// Axis Errors -----------------------------------------------------------------------------------------------------


17152   : sNcError := '17152 Parameter: Axis ID not allowed. The axis ID value is not allowed, e.g. because it has already been assigned, is out of the valid range [1 ... 255], or does not exist in the current configuration.';
17153   : sNcError := '17153 Parameter: Axis type not allowed. The axis type value is not allowed as it is not defined. Valid types: 1 (servo), 2 (fast/creep), 3 (stepper motor).';
17158   : sNcError := '17158 Parameter: Slow manual velocity not allowed. The slow manual velocity value is not allowed. Valid range: [0.0, 10000.0] e.g., m/min.';
17159   : sNcError := '17159 Parameter: Fast manual velocity not allowed. The fast manual velocity value is not allowed. Valid range: [0.0, 10000.0] e.g., m/min.';
17160   : sNcError := '17160 Parameter: Rapid traverse velocity not allowed. The rapid traverse velocity value is not allowed. Valid range: [0.0, 10000.0] e.g., m/min.';
17161   : sNcError := '17161 Parameter: Axis acceleration not allowed. The axis acceleration value is not allowed. Valid range: [0.0, 1000000.0] e.g., m/s².';
17162   : sNcError := '17162 Parameter: Axis deceleration not allowed. The axis deceleration value is not allowed. Valid range: [0.0, 1000000.0] e.g., m/s².';
17163   : sNcError := '17163 Parameter: Axis jerk not allowed. The axis jerk value is not allowed. Valid range: [0.0, 1000000.0] e.g., m/s³.';
17164   : sNcError := '17164 Parameter: Delay time between position and velocity not allowed. The delay time for dead time compensation is not allowed. Valid range: [0, 0.1] s.';
17165   : sNcError := '17165 Parameter: Override type not allowed. The velocity override type value is not allowed as it is not defined. Valid types: 1 (internal), 2 (external).';
17166   : sNcError := '17166 Parameter: NCI: Velo-Jump-Factor not allowed. The velo-jump-factor value is not allowed for TwinCAT NCI. Valid range: [0, 1000000].';
17167   : sNcError := '17167 Parameter: NCI: Tolerance sphere radius invalid. The tolerance sphere size value for auxiliary axes is invalid. Valid range: [0, 1000] e.g., mm.';
17168   : sNcError := '17168 Parameter: NCI: Max deviation for auxiliary axis invalid. The max allowed deviation value for auxiliary axes is invalid. Valid range: [0, 10000] e.g., mm.';
17170   : sNcError := '17170 Parameter: Referencing velocity in direction of cam not allowed. The referencing velocity towards the cam is not allowed. Valid range: [0.0, 10000.0] e.g., m/min.';
17171   : sNcError := '17171 Parameter: Referencing velocity in sync direction not allowed. The referencing velocity towards the sync pulse is not allowed. Valid range: [0.0, 10000.0] e.g., m/min.';
17172   : sNcError := '17172 Parameter: Pulse width in positive direction not allowed. The pulse width in the positive direction is not allowed for pulsed operation. Valid range: [0.0, 1000000.0] e.g., mm.';
17173   : sNcError := '17173 Parameter: Pulse width in negative direction not allowed. The pulse width in the negative direction is not allowed for pulsed operation. Valid range: [0.0, 1000000.0] e.g., mm.';
17174   : sNcError := '17174 Parameter: Pulse time in positive direction not allowed. The pulse time in the positive direction is not allowed. Valid range: [0.0, 600.0] s.';
17175   : sNcError := '17175 Parameter: Pulse time in negative direction not allowed. The pulse time in the negative direction is not allowed. Valid range: [0.0, 600.0] s.';
17176   : sNcError := '17176 Parameter: Creep distance in positive direction not allowed. The creep distance in the positive direction is not allowed. Valid range: [0.0, 100000.0] e.g., mm.';
17177   : sNcError := '17177 Parameter: Creep distance in negative direction not allowed. The creep distance in the negative direction is not allowed. Valid range: [0.0, 100000.0] e.g., mm.';
17178   : sNcError := '17178 Parameter: Braking distance in positive direction not allowed. The braking distance in the positive direction is not allowed. Valid range: [0.0, 100000.0] e.g., mm.';
17179   : sNcError := '17179 Parameter: Braking distance in negative direction not allowed. The braking distance in the negative direction is not allowed. Valid range: [0.0, 100000.0] e.g., mm.';
17180   : sNcError := '17180 Parameter: Deceleration time in positive direction not allowed. The deceleration time in the positive direction is not allowed. Valid range: [0.0, 60.0] s.';
17181   : sNcError := '17181 Parameter: Deceleration time in negative direction not allowed. The deceleration time in the negative direction is not allowed. Valid range: [0.0, 60.0] s.';
17182   : sNcError := '17182 Parameter: Switching time from rapid to slow traverse not allowed. The switching time from rapid to slow traverse is not allowed. Valid range: [0.0, 60.0] s.';
17183   : sNcError := '17183 Parameter: Creep distance for stop not allowed. The creep distance for an explicit stop is not allowed. Valid range: [0.0, 100000.0] e.g., mm.';
17184   : sNcError := '17184 Parameter: Motion monitoring not allowed. The motion monitoring activation value is not allowed. Valid range: [0, 1].';
17185   : sNcError := '17185 Parameter: Position window monitoring not allowed. The position window monitoring activation value is not allowed. Valid range: [0, 1].';
17186   : sNcError := '17186 Parameter: Target window monitoring not allowed. The target window monitoring activation value is not allowed. Valid range: [0, 1].';
17187   : sNcError := '17187 Parameter: Loop not allowed. The loop movement activation value is not allowed. Valid range: [0, 1].';
17188   : sNcError := '17188 Parameter: Motion monitoring time not allowed. The motion monitoring time value is not allowed. Valid range: [0.0, 600.0] s.';
17189   : sNcError := '17189 Parameter: Target window range not allowed. The target window value is not allowed. Valid range: [0.0, 10000.0] e.g., mm.';
17190   : sNcError := '17190 Parameter: Position window range not allowed. The position window value is not allowed. Valid range: [0.0, 10000.0] e.g., mm.';
17191   : sNcError := '17191 Parameter: Position window monitoring time not allowed. The position window monitoring time value is not allowed. Valid range: [0.0, 600.0] s.';
17192   : sNcError := '17192 Parameter: Looping distance not allowed. The looping distance value is not allowed. Valid range: [0.0, 10000.0] e.g., mm.';
17193   : sNcError := '17193 Parameter: Axis cycle time not allowed. The axis cycle time value is not allowed. Valid range: [0.001, 0.1] s.';
17194   : sNcError := '17194 Parameter: Operation mode stepper motor not allowed. The stepper motor operating mode value is not allowed. Valid range: [1, 2].';
17195   : sNcError := '17195 Parameter: Displacement per stepper motor step not allowed. The displacement per step value for the stepper motor is not allowed. Valid range: [0.000001, 1000.0] e.g., mm/STEP.';
17196   : sNcError := '17196 Parameter: Minimum velocity for stepper motor set value profile not allowed. The minimum velocity for the stepper motor velocity profile is not allowed. Valid range: [0.0, 1000.0] e.g., m/min.';
17197   : sNcError := '17197 Parameter: Stepper motor stages for one velocity level not allowed. The number of steps for each velocity level in the setpoint generation is not allowed. Valid range: [0, 100].';
17198   : sNcError := '17198 Parameter: DWORD for the interpretation of the axis units not allowed. The flags value for interpreting position and velocity units is not allowed. Valid range: [0, 0xFFFFFFFF].';
17199   : sNcError := '17199 Parameter: Maximum velocity not allowed. The maximum permitted velocity value is not allowed. Valid range: [0.0, 10000.0] e.g., m/min.';
17200   : sNcError := '17200 Parameter: Motion monitoring window not allowed. The motion monitoring window value is not allowed. Valid range: [0.0, 10000.0] e.g., mm.';
17201   : sNcError := '17201 Parameter: PEH time monitoring not allowed. The PEH time monitoring activation value is not allowed (PEH: positioning end and halt). Valid range: [0, 1].';
17202   : sNcError := '17202 Parameter: PEH monitoring time not allowed. The PEH monitoring time (timeout) value is not allowed (PEH: positioning end and halt). Valid range: [0.0, 600.0] s.';
17203   : sNcError := '17203 Parameter: Brake Release Delay is invalid. The brake release delay parameter for a rapid/slow traverse axis is invalid. Valid range: [0.0, 60.0] s.';
17204   : sNcError := '17204 Parameter: NC Data Persistence is invalid. The boolean parameter NC Data Persistence of an axis is invalid. Valid range: [0, 1].';
17205   : sNcError := '17205 Parameter: Error reaction mode is invalid. The error reaction mode parameter of the axis is invalid (instantaneous, delayed). Valid range: [0, 1].';
17206   : sNcError := '17206 Parameter: Error reaction delay is invalid. The error reaction delay parameter of the axis is invalid. Valid range: [0.0, 1000.0] s.';
17207   : sNcError := '17207 Parameter: Use actual values in deactivated state is invalid. The parameter "Use actual values in deactivated state" is invalid. Valid range: [0, 1].';
17208   : sNcError := '17208 Parameter: Allow motion commands for slave axes is invalid. The boolean parameter "Allow motion commands for slave axes" is invalid. Valid range: [0, 1].';
17209   : sNcError := '17209 Parameter: Allow motion commands for axis in external setpoint generation is invalid. The boolean parameter "Allow motion commands for axis in external setpoint generation" is invalid. Valid range: [0, 1].';
17210   : sNcError := '17210 Parameter: Fading Acceleration is invalid. The "Fading Acceleration" parameter for the fading profile from SET to ACTUAL values is invalid. Valid range: [0; 0.01 .. 1.0e+20] e.g., mm/s².';
17211   : sNcError := '17211 Parameter: Fast Axis Stop signal type not allowed. The Signal Type value of the "Fast Axis Stop" is not allowed. Valid range: [0...5].';
17212   : sNcError := '17212 Parameter: ADS index offset not allowed. The "ADS offset (axis state)" value for user-defined parameter named "UserData" in AxisRef is invalid.';
17216   : sNcError := '17216 Initialization: Axis initialization. The axis has not been fully initialized (I/O, axis, reset).';
17217   : sNcError := '17217 Address: Group address. The axis does not have a group or the group address has not been initialized.';
17218   : sNcError := '17218 Address: Encoder address. The axis does not have an encoder or the encoder address has not been initialized.';
17219   : sNcError := '17219 Address: Controller address. The axis does not have a controller or the controller address has not been initialized.';
17220   : sNcError := '17220 Address: Drive address. The axis does not have a drive or the drive address has not been initialized.';
17221   : sNcError := '17221 Address: Axis interface PLC to NC address. The axis has no axis interface from the PLC to the NC (PlcToNc) or the axis interface address has not been initialized.';


// Drive Errors -----------------------------------------------------------------------------------------------------


17920   : sNcError := '17920 Parameter: Drive ID not allowed. The drive ID value is invalid because it is either already assigned, less than or equal to zero, or exceeds 255. Valid range: [1 ... 255].';
17921   : sNcError := '17921 Parameter: Drive type not allowed. The drive type value is invalid as it is not defined. Valid range: [1, 20].';
17922   : sNcError := '17922 Parameter: Drive operation mode not allowed. The drive operation mode value is invalid. Valid range: [1].';
17923   : sNcError := '17923 Parameter: Motor polarity not allowed. The motor polarity flag is invalid. Valid values: 0 (Positive), 1 (Negative).';
17924   : sNcError := '17924 Parameter: Drift compensation/velocity offset (DAC offset) invalid. Valid range: [-100.0, 100.0] e.g., m/min.';
17925   : sNcError := '17925 Parameter: Reference velocity (velocity pre-control) invalid. Valid range: [0.0, 10000.0] e.g., m/min.';
17926   : sNcError := '17926 Parameter: Reference output in percent invalid. The value usually corresponds to a voltage of 10.0 V. Valid range: [0.0, 5.0] %.';
17927   : sNcError := '17927 Parameter: Quadrant compensation factor not allowed. The value is invalid. Valid range: [0.0, 100.0].';
17928   : sNcError := '17928 Parameter: Velocity reference point in percent invalid. The value 1.0 corresponds to 100 percent. Valid range: [0.01, 1.0] %.';
17929   : sNcError := '17929 Parameter: Output reference point invalid. The value 1.0 corresponds to 100 percent. Valid range: [0.01, 1.0] %.';
17930   : sNcError := '17930 Parameter: Min or max output limits (output limitation) invalid. The min limit is initially set to –1.0 (-100%) and the max limit to 1.0 (100%). Valid range: [-1.0, 1.0] %.';
17931   : sNcError := '17931 Parameter: Maximum value for output not allowed. The value for the max output digits of the drive is not allowed. Valid range: [0x000000FF .. 0xFFFFFFFF] INC or Digits.';
17932   : sNcError := '17932 Parameter: Internal Drive Control Word not allowed. The internal Drive Control Word value for the NC is invalid. Valid range: [>0].';
17933   : sNcError := '17933 Parameter: Internal timer for RESET behavior Drive not allowed. The timer influencing NC Drive and IO Drive behavior is invalid. Valid range: [>5] NC SEC cycles.';
17934   : sNcError := '17934 Parameter: Master Motion Controller ID not allowed. This parameter is invalid for a slave NC Motion Controller. Valid range: [0 .. 255].';
17935   : sNcError := '17935 Parameter: Drive torque output scaling not allowed. The value for Drive torque output scaling (rotary motor) or force output scaling (linear motor) is invalid. Valid range: [0, 1000000].';
17936   : sNcError := '17936 Parameter: Drive velocity output scaling not allowed. The value is invalid. Valid range: [0, 1000000].';
17937   : sNcError := '17937 Parameter: Profi Drive DSC proportional gain Kpc (controller) not allowed. The Profi Drive DSC position control gain (Kpc factor) value is invalid. Valid range: [0, 0xFFFFFF] 0.001 * 1/s.';
17938   : sNcError := '17938 Parameter: Table ID not allowed. The table ID value is invalid. Valid range: [0, 255].';
17939   : sNcError := '17939 Parameter: Table interpolation type not allowed. The table interpolation type value is invalid. Valid values: 0 (LINEAR), 2 (SPLINE).';
17940   : sNcError := '17940 Parameter: Output offset in percent not allowed. The output offset in percent value is invalid. Valid range: [-1.0, 1.0] %.';
17941   : sNcError := '17941 Parameter: Profi Drive DSC scaling for "Xerr" (controller) not allowed. The value is invalid. Valid range: [0, 1000000].';
17942   : sNcError := '17942 Parameter: Drive acceleration output scaling not allowed. The value is invalid. Valid range: [0, 1000000].';
17943   : sNcError := '17943 Parameter: Drive position output scaling not allowed. The value is invalid. Valid range: [0, 1000000].';
17944   : sNcError := '17944 Parameter: Dead time compensation mode (Motion Controller) invalid. The dead time compensation mode is invalid (OFF, ON with velocity, ON with velocity and acceleration). Valid values: [0, 1, 2].';
17945   : sNcError := '17945 Parameter: Control bits of dead time compensation (motion controller) invalid. The parameter is invalid. Valid range: [>0].';
17946   : sNcError := '17946 Parameter: Time shift of dead time compensation mode (motion controller) invalid. The time shift parameter in nanoseconds is invalid. Valid range: [-1.0E9 .. 1.0E9] ns.';
17947   : sNcError := '17947 Parameter: Output delay velocity interface Motion Controller invalid. The optional output delay in the velocity interface is invalid. Valid range: [0.0 .. 0.1] s.';
17948   : sNcError := '17948 Parameter: Drive filter type not allowed for command variable filter for the output position. The drive filter type value is invalid. Valid range: [0, 2].';
17949   : sNcError := '17949 Parameter: Drive filter time not allowed for command variable filter for the output position. The drive filter time value is invalid. Valid range: [0.0, 1.0] s.';
17950   : sNcError := '17950 Parameter: Drive filter order not allowed for command variable filter for the output position. The drive filter order value is invalid. Valid range: [0, 10].';
17952   : sNcError := '17952 Parameter: Bit mask for stepper motor cycle not allowed. The bit mask value is invalid. Valid range: [0, 255].';
17953   : sNcError := '17953 Parameter: Bit mask for stepper motor holding current not allowed. The holding current mask value is invalid. Valid range: [0, 255].';
17954   : sNcError := '17954 Parameter: Scaling factor for actual torque (actual current) not allowed. The scaling factor value is invalid. Valid range: [0, 1E+30].';
17955   : sNcError := '17955 Parameter: Filter time for actual torque not allowed. The filter time value for the actual torque (or current) is invalid. Valid range: [0.0, 60.0] s.';
17956   : sNcError := '17956 Parameter: Filter time for the time derivative of the actual torque not allowed. The filter time value for the time derivative of the actual torque (or current) is invalid. Valid range: [0.0, 60.0] s.';
17957   : sNcError := '17957 Parameter: Drive operation mode invalid. The drive operation mode parameter is invalid. Valid range: [0, >=1].';
17958   : sNcError := '17958 Monitoring: Motion Controller function not supported. The triggered Motion Controller functionality is not enabled or implemented.';
17959   : sNcError := '17959 Function: DRIVEOPERATIONMODEBUSY. The drive operation mode activation failed because another object is using this interface.';
17960   : sNcError := '17960 Monitoring: Drive operation mode changeover not configured. No drive operation mode changeover is configured or the desired mode is not found.';
17961   : sNcError := '17961 Monitoring: Feedback drive operation mode changeover. The requested drive operation mode was not consistently reported back within the monitoring time.';
17968   : sNcError := '17968 Monitoring: Overtemperature detected or reported in the drive or terminal.';
17969   : sNcError := '17969 Monitoring: Undervoltage detected or reported in the drive or terminal.';
17970   : sNcError := '17970 Monitoring: Wire break in phase A detected or reported in the drive or terminal.';
17971   : sNcError := '17971 Monitoring: Wire break in phase B detected or reported in the drive or terminal.';
17972   : sNcError := '17972 Monitoring: Overcurrent detected or reported in phase A in the drive or terminal.';
17973   : sNcError := '17973 Monitoring: Overcurrent detected or reported in phase B in the drive or terminal.';
17974   : sNcError := '17974 Monitoring: Torque overload (stall) detected or reported in the drive or terminal.';
17984   : sNcError := '17984 Initialization: Drive initialization. Drive not initialized properly. Steps: 1. Initialization drive I/O, 2. Initialization drive, 3. Reset drive.';
17985   : sNcError := '17985 Address: Axis address not initialized. The drive does not know its axis or the axis address is not initialized.';
17986   : sNcError := '17986 Address: Address I/O input structure. The drive has no valid I/O input address in the process image.';
17987   : sNcError := '17987 Address: Address I/O output structure. The drive has no valid I/O output address in the process image.';
18000   : sNcError := '18000 Monitoring: Drive hardware not ready. The drive hardware is not ready for operation, possibly due to hardware error, start-up phase, or missing controller enable.';
18001   : sNcError := '18001 Monitoring: Error in cyclic communication of the drive (Life Counter). Possible causes: interrupted fieldbus or drive in error state.';
18002   : sNcError := '18002 Monitoring: Changing table ID with active controller enable not allowed. Changing the characteristic curve table ID is not allowed when controller enable is active.';
18005   : sNcError := '18005 Monitoring: I/O data for more than "n" continuous NC cycles invalid. The axis detected invalid I/O data for more than "n" continuous NC cycles.';


// Controller Errors -----------------------------------------------------------------------------------------------------


17664   : sNcError := '17664 Parameter: Controller ID not allowed. The controller ID value is invalid, e.g., already assigned, less than or equal to zero, or exceeds 255. Valid range: [1 ... 255].';
17665   : sNcError := '17665 Parameter: Controller type not allowed. The controller type value is invalid as it is not defined. Valid types: 1 (P-controller), 7 (Fast/creep), 8 (Stepper motor), 9 (Sercos).';
17666   : sNcError := '17666 Parameter: Operation mode controller not allowed. The controller operating mode value is invalid. Valid range: [1].';
17667   : sNcError := '17667 Parameter: Weighting of the velocity pre-control not allowed. The velocity pre-control weighting value is invalid. Valid range: [0.0 ... 1.0] %.';
17668   : sNcError := '17668 Parameter: Lag error monitor (position) not allowed. The activation value for the lag error monitor is invalid. Valid range: [0, 1].';
17669   : sNcError := '17669 Parameter: Lag monitoring (velocity) not allowed. The activation value for the lag error monitoring is invalid. Valid range: [0, 1].';
17670   : sNcError := '17670 Parameter: Lag error window (position) not allowed. The maximum allowable lag error value is invalid. Valid range: [0.0, 10000.0] e.g., mm.';
17671   : sNcError := '17671 Parameter: Lag error filter time (position) not allowed. The lag error filter time value is invalid. Valid range: [0.0, 600.0] s.';
17672   : sNcError := '17672 Parameter: Lag error window (velocity) not allowed. The lag error window (velocity) value is invalid. Valid range: [0.0, 10000.0] e.g., m/min.';
17673   : sNcError := '17673 Parameter: Lag error filter time (velocity) not allowed. The lag error filter time value is invalid. Valid range: [0.0, 600.0] s.';
17674   : sNcError := '17674 Parameter: Controller output limitation not allowed. The output limitation value of the controller is invalid. Valid range: [0.0, 1.0] %.';
17680   : sNcError := '17680 Parameter: Proportional gain Kv or Kp (controller) not allowed. The proportional gain (Kv or Kp factor) value is invalid. Valid range: [0.0, 10000.0] e.g., mm/s/mm.';
17681   : sNcError := '17681 Parameter: Integral action time Tn (controller) not allowed. The integral action time value is invalid (I part of the PID T1 controller). Valid range: [0.0, 60.0] s.';
17682   : sNcError := '17682 Parameter: Rate time Tv (controller) not allowed. The derivative action time value is invalid (D part of the PID T1 controller). Valid range: [0.0, 60.0] s.';
17683   : sNcError := '17683 Parameter: Damping time Td (controller) not allowed. The damping time value is invalid (D part of the PID T1 controller). Valid range: [0.0, 60.0] s.';
17684   : sNcError := '17684 Function: Activation of the automatic offset calibration not allowed. Activation of automatic offset calibration is only possible for certain controllers (without I component).';
17685   : sNcError := '17685 Parameter: Additional proportional gain Kv or Kp (controller) not allowed. The second term of the proportional gain value is invalid. Valid range: [0.0, 10000.0] e.g., mm/s/mm.';
17686   : sNcError := '17686 Parameter: Reference velocity for additional proportional gain Kv or Kp (controller) not allowed. The reference velocity percentage value is invalid. Standard: 0.5 (50%). Valid range: [0.0 ... 1.0] %.';
17687   : sNcError := '17687 Parameter: Proportional gain Pa (proportion) not allowed. The proportional gain (Pa factor) value is invalid. Valid range: [0.0, 1000000.0] s.';
17688   : sNcError := '17688 Parameter: Proportional gain Kv (controller) not allowed. The proportional gain (Kv factor) value is invalid. Valid range: [0.0, 10000.0].';
17689   : sNcError := '17689 Parameter: Integral action time Tn (controller) not allowed. The integral action time value is invalid (I part of the PID T1 controller). Valid range: [0.0, 60.0] s.';
17690   : sNcError := '17690 Parameter: Reserved. Reserved, currently not used.';
17691   : sNcError := '17691 Parameter: Reserved. Reserved, currently not used.';
17692   : sNcError := '17692 Parameter: Velocity filter time not allowed. The velocity filter time in seconds (P-T1 filter) is invalid. Valid range: [0.0, 60.0] s.';
17693   : sNcError := '17693 Parameter: Dead range not allowed. The dead range (neutral zone) value of the position or velocity error is invalid. Valid range: [0.0, 10000.0] mm or mm/s.';
17695   : sNcError := '17695 Parameter: Proportional gain Kcp not allowed. The proportional gain Kcp parameter for slave coupling difference control is invalid. Valid range: [0.0, 10000.0] e.g., mm²/mm.';
17696   : sNcError := '17696 Parameter: Rate time Tv (controller) not allowed. The derivative action time value is invalid (D part of the PID T1 controller). Valid range: [0.0, 60.0] s.';
17697   : sNcError := '17697 Parameter: Damping time Td (controller) not allowed. The damping time value is invalid (D part of the PID T1 controller). Valid range: [0.0, 60.0] s.';
17698   : sNcError := '17698 Parameter: Limitation of the I part not allowed. The limitation parameter for the I-part of a PI- or PID-controller is invalid. Valid range: [0.0 .. 1.0] %.';
17699   : sNcError := '17699 Parameter: Limitation of the D part not allowed. The limitation parameter for the D-part of a PI- or PID-controller is invalid. Valid range: [0.0 .. 1.0] %.';
17700   : sNcError := '17700 Parameter: Deactivation of the I part during travel not allowed. The boolean parameter for switching off the I-part during active positioning is invalid. Valid range: [0, 1].';
17701   : sNcError := '17701 Parameter: Filter time for P-T2 filter not allowed. The filter time T0 for the P-T2 element is invalid. Valid range: [0.0, 60.0] s.';
17702   : sNcError := '17702 Parameter: Velocity observer mode not allowed. The parameterized mode (0=OFF, 1=LUENBERGER) for the velocity observer is invalid. Valid range: [0, 1].';
17703   : sNcError := '17703 Parameter: Motor torque constant Kt or Kf not allowed. The motor torque constant Kt (rotary) or Kf (linear) parameter for the velocity observer is invalid. Valid range: [0.0 .. 100000.0] Nm/A or N/A.';
17704   : sNcError := '17704 Parameter: Motor moment of inertia JM not allowed. The motor moment of inertia JM parameter for the velocity observer is invalid. Valid range: [0.0001 .. 100000.0] kg cm².';
17705   : sNcError := '17705 Parameter: Bandwidth f0 not allowed. The bandwidth f0 parameter for the velocity observer is invalid. Valid range: [0.0 .. 10000.0] Hz.';
17706   : sNcError := '17706 Parameter: Correction factor kc not allowed. The correction factor kc for the velocity observer is invalid. Valid range: [0.0 .. 100.0] s.';
17707   : sNcError := '17707 Parameter: Time constant T for 1st order filter not allowed. The time constant T for the 1st order velocity filter is invalid. Valid range: [0.0 .. 100.0] s.';
17708   : sNcError := '17708 Parameter: Amplitude damping d for 2nd order filter not allowed. The amplitude damping dHP or dTP for the 2nd order filter is invalid. Valid range: [0.2 .. 10.0].';
17709   : sNcError := '17709 Parameter: Frequency fHP or fTP for 2nd order filter not allowed. The frequency fHP or fTP for the 2nd order filter is invalid. Valid range: [0.0 .. 10000.0] Hz.';
17728   : sNcError := '17728 Initialization: Controller initialization. The controller has not been initialized properly. Steps: 1. Initialization of controller, 2. Reset of controller.';
17729   : sNcError := '17729 Address: Axis address not initialized. The controller does not know its axis or the axis address is not initialized.';
17730   : sNcError := '17730 Address: Drive address not initialized. The controller does not know its drive or the drive address is not initialized.';
17744   : sNcError := '17744 Monitoring: Lag error monitor (position). The lag error exceeded the window and lasted longer than the filter time during lag error monitor activation.';
17745   : sNcError := '17745 Monitoring: Lag monitoring (velocity). The velocity lag error exceeded the window and lasted longer than the filter time during lag error monitor activation.';
17824   : sNcError := '17824 Monitoring: Internal error. CONTROLERR_RANGE_AREA_ASIDE.';
17825   : sNcError := '17825 Monitoring: Internal error. CONTROLERR_RANGE_AREA_BSIDE.';
17826   : sNcError := '17826 Monitoring: Internal error. CONTROLERR_RANGE_QNENN.';
17827   : sNcError := '17827 Monitoring: Internal error. CONTROLERR_RANGE_PNENN.';
17828   : sNcError := '17828 Monitoring: Internal error. CONTROLERR_RANGE_AXISIDPRESP0.';


// Encoder Errors -----------------------------------------------------------------------------------------------------


17408   : sNcError := '17408 Parameter: Encoder ID not allowed. The encoder ID value is invalid because it is already assigned, less than or equal to zero, or exceeds 255. Valid range: [1 ... 255].';
17409   : sNcError := '17409 Parameter: Encoder type not allowed. The encoder type value is invalid as it is not defined. Valid types: 1 (Simulation), 2 (M3000), 3 (M31x0), 4 (KL5101), 5 (KL5001), 6 (KL5051).';
17410   : sNcError := '17410 Parameter: Encoder mode not allowed. The encoder operation mode value is invalid. Valid modes: 1 (Position), 2 (Position and velocity).';
17411   : sNcError := '17411 Parameter: Encoder count direction not allowed. The encoder counting direction flag is invalid. Valid values: 0 (Positive), 1 (Negative).';
17412   : sNcError := '17412 Initialization: Calibration state not allowed. The calibration state flag is invalid. Valid values: 0 (Not referenced), 1 (Referenced).';
17413   : sNcError := '17413 Parameter: Encoder increments per revolution not allowed. The number of encoder increments per revolution is invalid. Valid range: [255, 0xFFFFFFFF] INC.';
17414   : sNcError := '17414 Parameter: Scaling factor not allowed. The scaling factor for converting encoder increments to physical units is invalid. Valid range: [0.000001, 100.0] e.g., mm/INC.';
17415   : sNcError := '17415 Parameter: Position offset not allowed. The position offset value is invalid. Valid range: [-1000000.0, 1000000.0] e.g., mm.';
17416   : sNcError := '17416 Parameter: Modulo factor not allowed. The modulo factor value is invalid. Valid range: [1.0, 1.0E+9] e.g., mm or degrees.';
17417   : sNcError := '17417 Parameter: Position filter time not allowed. The actual position filter time value is invalid (P-T1 filter). Valid range: [0.0, 60.0] s.';
17418   : sNcError := '17418 Parameter: Velocity filter time not allowed. The actual velocity filter time value is invalid (P-T1 filter). Valid range: [0.0, 60.0] s.';
17419   : sNcError := '17419 Parameter: Acceleration filter time not allowed. The actual acceleration filter time value is invalid (P-T1 filter). Valid range: [0.0, 60.0] s.';
17420   : sNcError := '17420 Initialization: Cycle time not allowed (internal error). The SAF cycle time value for actual values calculation is invalid.';
17421   : sNcError := '17421 Initialization: Setting of selected units is invalid. Settings for modulo position, velocity, etc., lead to an error.';
17422   : sNcError := '17422 Parameter: Position correction/measurement system error correction not allowed. The activation value for actual position correction is invalid. Valid range: [0, 1].';
17423   : sNcError := '17423 Parameter: Position correction filter time not allowed. The filter time value for actual position correction is invalid (P-T1 filter). Valid range: [0.0, 60.0] s.';
17424   : sNcError := '17424 Parameter: Search direction for referencing cam inverted. The search direction value for the referencing cam is invalid. Valid values: 0 (Positive), 1 (Negative).';
17425   : sNcError := '17425 Parameter: Search direction for sync pulse inverted. The search direction value for the sync pulse is invalid. Valid values: 0 (Positive), 1 (Negative).';
17426   : sNcError := '17426 Parameter: Reference position not allowed. The reference position value in a referencing procedure is invalid. Valid range: [-1000000.0, 1000000.0] e.g., mm.';
17427   : sNcError := '17427 Parameter: Distance monitoring between hardware latch activation and sync pulse occurrence not allowed. The distance monitoring flag is invalid. Valid values: 0 (Passive), 1 (Active).';
17428   : sNcError := '17428 Parameter: Minimum gap between hardware latch activation and sync pulse not allowed. The minimum gap value between hardware latch activation and sync pulse is invalid. Valid range: [0, 65536] INC.';
17429   : sNcError := '17429 Parameter: External sync pulse not allowed. The activation/deactivation value for the external sync pulse is invalid. Valid values: 0 (Passive), 1 (Active).';
17430   : sNcError := '17430 Parameter: Scaling of the noise rate not allowed. The scaling value for the synthetic noise rate is invalid. Valid range: [0, 1000000].';
17431   : sNcError := '17431 Parameter: Tolerance window for modulo-start not allowed. The tolerance window value for the modulo-axis-start is invalid. Valid range: [0.0, 180.0] e.g., mm or degrees.';
17432   : sNcError := '17432 Parameter: Encoder referencing mode not allowed. The encoder referencing mode value is invalid or unsupported. Valid range: [0, 5].';
17433   : sNcError := '17433 Parameter: Encoder evaluation direction not allowed. The encoder evaluation direction value is invalid. Valid range: [0, 3].';
17434   : sNcError := '17434 Parameter: Encoder absolute dimensioning system not allowed. The encoder reference system value is invalid. Valid values: 0 (INCREMENTAL), 1 (ABSOLUTE), 2 (ABSOLUTE+MODULO).';
17435   : sNcError := '17435 Parameter: Encoder position initialization mode not allowed. The encoder position initialization mode value at TC system startup is invalid. Valid range: [0, 1].';
17436   : sNcError := '17436 Parameter: Encoder sign interpretation (UNSIGNED/SIGNED) not allowed. The encoder sign interpretation value is invalid. Valid values: 0 (Default), 1 (UNSIGNED), 2 (SIGNED).';
17437   : sNcError := '17437 Parameter: Homing Sensor Source not allowed. The Encoder Homing Sensor Source value is invalid or unsupported. Valid range: [0, 16].';
17440   : sNcError := '17440 Parameter: Software end position monitoring minimum not allowed. The activation value for software end position monitoring minimum is invalid. Valid range: [0, 1].';
17441   : sNcError := '17441 Parameter: Software end position monitoring maximum not allowed. The activation value for software end position monitoring maximum is invalid. Valid range: [0, 1].';
17442   : sNcError := '17442 Function: Actual value setting outside value range. The "Set actual value" function cannot be executed as the new position is outside the intended value range. Valid range: [-1.0E10, 1.0E10] e.g., mm.';
17443   : sNcError := '17443 Parameter: Software end position minimum not allowed. The software end position minimum value is invalid. Valid range: [-1000000000.0, 1000000000.0] e.g., mm.';
17444   : sNcError := '17444 Parameter: Software end position maximum not allowed. The software end position maximum value is invalid. Valid range: [-1000000000.0, 1000000000.0] e.g., mm.';
17445   : sNcError := '17445 Parameter: Filter mask for encoder raw value not allowed. The filter mask value for the encoder raw value in increments is invalid. Valid range: [0x0, 0xFFFFFFFF].';
17446   : sNcError := '17446 Parameter: Reference mask for encoder raw value not allowed. The reference mask value for the encoder raw value in increments is invalid. Valid range: [0x0000000F, 0xFFFFFFFF].';
17447   : sNcError := '17447 Parameter: Dead time compensation mode (encoder) invalid. The dead time compensation mode on the NC encoder is invalid. Valid values: [0, 1, 2].';
17448   : sNcError := '17448 Parameter: Control bits of dead time compensation (encoder) invalid. The control bits value for dead time compensation at the encoder is invalid. Valid range: [>0].';
17449   : sNcError := '17449 Parameter: Time shift of dead time compensation mode (encoder) invalid. The time shift parameter for dead time compensation at the encoder is invalid. Valid range: [-1.0E9 .. 1.0E9] ns.';
17456   : sNcError := '17456 Function: Hardware latch activation (encoder). The encoder hardware latch activation was initiated by referencing. If already active and latch value not valid, another call is refused.';
17457   : sNcError := '17457 Function: Activation of external hardware latch/touch probe function (encoder). External hardware latch activation is invalid if already active without valid latch value.';
17458   : sNcError := '17458 Function: External hardware latch activation (encoder). Referencing procedure with valid latch value already active.';
17459   : sNcError := '17459 Function: Activation of external hardware latch/touch probe function (encoder). Function activated before and not finished, renewed activation not allowed.';
17460   : sNcError := '17460 Monitoring: Encoder function not supported. An unsupported or not released encoder function has been activated.';
17461   : sNcError := '17461 Monitoring: Encoder function already active. Encoder function cannot be activated as it is already active.';
17472   : sNcError := '17472 Initialization: Encoder initialization not completed. Steps: 1. Initialization of axis I/O, 2. Initialization of axis, 3. Reset axis.';
17473   : sNcError := '17473 Address: Axis address not initialized. The encoder does not know its axis or the axis address is not initialized.';
17474   : sNcError := '17474 Address: Address I/O input structure invalid. The drive has no valid I/O input address in the process image.';
17475   : sNcError := '17475 Address: Address I/O output structure invalid. The encoder has no valid I/O output address in the process image.';
17488   : sNcError := '17488 Monitoring: Encoder counter underflow detected.';
17489   : sNcError := '17489 Monitoring: Encoder counter overflow detected.';
17504   : sNcError := '17504 Monitoring: Minimum software position limit (axis start). Axis start below the minimum software position limit detected.';
17505   : sNcError := '17505 Monitoring: Maximum software position limit (axis start). Axis start above the maximum software position limit detected.';
17506   : sNcError := '17506 Monitoring: Minimum software position limit (positioning process). Actual position fell below the minimum software position limit.';
17507   : sNcError := '17507 Monitoring: Maximum software position limit (positioning process). Actual position exceeded the maximum software position limit.';
17508   : sNcError := '17508 Monitoring: Encoder hardware error reported by drive or encoder system.';
17509   : sNcError := '17509 Monitoring: Position initialization error at system startup. Actual position outside min/max end positions for all three initialization attempts.';
17510   : sNcError := '17510 Monitoring: Invalid I/O data for more than "n" NC cycles (encoder). Invalid encoder I/O data detected for more than "n" continuous NC cycles.';
17511   : sNcError := '17511 Monitoring: Invalid actual position (encoder). I/O device returns an invalid actual position.';
17512   : sNcError := '17512 Monitoring: Invalid I/O input data (error type 1). Cyclic I/O input counter error detected (data not updated for 3 NC-SAF cycles).';
17513   : sNcError := '17513 Monitoring: Invalid I/O input data (error type 2). Cyclic I/O input counter error detected (insufficient data quality based on 2-bit counter).';
17520   : sNcError := '17520 Monitoring: SSI transformation faulty or not finished. SSI transformation of the FOX 50 module was faulty for some NC-cycles or did not finish.';
17570   : sNcError := '17570 Monitoring: Internal error. ENCERR_ADDR_CONTROLLER.';
17571   : sNcError := '17571 Monitoring: Internal error. ENCERR_INVALID_CONTROLLERTYPE.';


// Futher Errors -----------------------------------------------------------------------------------------------------


33056   : sNcError := '33056 Environment: Invalid configuration for Object (e.g. in TwinCAT 3 Engineering (XAE)).';
33057   : sNcError := '33057 Environment: Invalid environment for Object (e.g. TcCom-Object\s Hierarchy or missing/faulty Objects).';
33058   : sNcError := '33058 Environment: Incompatible Driver or Object.';
33060   : sNcError := '33060 Function Block: Command execution does not terminate (e.g. MC_Reset does not signal DONE).';
33072   : sNcError := '33072 Communication: Invalid ObjectID of Communication Target.';
33073   : sNcError := '33073 Communication: Communication Target expects Call in different Context.';
33074   : sNcError := '33074 Communication: Invalid State of Communication Target.';
33076   : sNcError := '33076 Communication: Communication with Communication Target cannot be established.';
33083   : sNcError := '33083 Parameter: Transition Mode is invalid.';
33084   : sNcError := '33084 Parameter: BufferMode is invalid.';
33085   : sNcError := '33085 Function Block: Only one active Instance of Function Block per Group is allowed.';
33086   : sNcError := '33086 State: Command is not allowed in current group state.';
33087   : sNcError := '33087 Function Block: Slave cannot synchronize. The slave cannot reach the SlaveSyncPosition with the given dynamics.';
33088   : sNcError := '33088 Parameter: Invalid value for one or more dynamic parameters (Acceleration, Deceleration, Jerk).';
33089   : sNcError := '33089 Parameter: IdentInGroup is invalid.';
33090   : sNcError := '33090 Parameter: Number of axes in the group incompatible with axes convention.';
33091   : sNcError := '33091 Communication: Function Block or Command not supported by Target.';
33092   : sNcError := '33092 State: Command queue full. Cannot accept more commands until some are fully processed.';
33093   : sNcError := '33093 Function Block: Mapping of Cyclic Interface between NC and PLC is missing (e.g. AXIS_REF, AXES_GROUP_REF, ...).';
33094   : sNcError := '33094 Function Block: Invalid Velocity Value. The velocity was not set or the entered value is invalid.';
33095   : sNcError := '33095 Parameter: Invalid Coordinate Dimension. The set coordinate interpretation does not meet requirements.';
33096   : sNcError := '33096 Function Block: Invalid Input Value.';
33097   : sNcError := '33097 Parameter: Unsupported Dynamics for selected Group Kernel.';
33098   : sNcError := '33098 Parameter: Programmed position dimension incompatible with axes convention.';
33099   : sNcError := '33099 Function Block: Path buffer is invalid (invalid address or too small).';
33100   : sNcError := '33100 Function Block: Path does not contain any element.';
33101   : sNcError := '33101 Function Block: Provided Path buffer too small for more Path Elements.';
33102   : sNcError := '33102 Parameter: Dimension or Value of Transition Parameters is invalid.';
33103   : sNcError := '33103 Function Block: Invalid or Incomplete Input Array.';
33104   : sNcError := '33104 Function Block: Path length is zero.';
33105   : sNcError := '33105 State: Command not allowed in current axis state.';
33106   : sNcError := '33106 State: TwinCAT System is shutting down and cannot complete request.';
33107   : sNcError := '33107 Parameter: Configured axes convention and configured axes do not match.';
33108   : sNcError := '33108 Initialization: Invalid Number of ACS Axes. The number of ACS input axes does not match expected by kinematic transformation.';
33109   : sNcError := '33109 Initialization: Invalid Number of MCS Data. The number of MCS input data does not match expected by kinematic transformation.';
33110   : sNcError := '33110 Initialization: Invalid Value Set for Kinematic Parameters. Value set for parameter is outside definition range.';
33112   : sNcError := '33112 NC Programming: Given ACS Values Cannot be Reached. Results in an invalid machine configuration.';
33113   : sNcError := '33113 NC Programming: Set Target Positions Cannot be Reached. Reside outside the admissible working space.';
33117   : sNcError := '33117 NC Programming: Discontinuity in ACS axes detected.';
33120   : sNcError := '33120 NC Programming: Circle Specification in Path is invalid. Circle segment specification in interpolated path has an invalid or ambiguous description.';
33121   : sNcError := '33121 NC Programming: Maximum stream lines reached. Refer to function block documentation for details.';
33123   : sNcError := '33123 Function Block: Invalid First Segment. Element can only be analyzed with a well-defined start point.';
33124   : sNcError := '33124 Function Block: Invalid auxiliary point. Auxiliary point is not well-defined.';
33126   : sNcError := '33126 Function Block: Invalid parameter for GapControlMode.';
33127   : sNcError := '33127 External: Group got unsupported Axis Event (e.g. State Change).';
33128   : sNcError := '33128 Parameter: Unsupported Compensation Type. Compensation type not set or unsupported by the object.';
33129   : sNcError := '33129 Function Block: Master axis does not exist or cannot be used.';
33130   : sNcError := '33130 External: Invalid or Missing Tracking Transformation. Invalid object ID or unsupported coordinate transformation at CoordTransform input.';
33131   : sNcError := '33131 Function Block: Position is not on Track. Actual or Target Position not on Track or TrackPart.';
33132   : sNcError := '33132 Function Block: Axis does not have an activated track.';
33133   : sNcError := '33133 NC Programming: Invalid Compensation ObjectId. Object with this ObjectId does not exist or is not of the right type.';
33134   : sNcError := '33134 Monitoring: Axis is in error because it was not in Target when InTargetAlarm Timer expired.';
33135   : sNcError := '33135 State: Coupling would cause a cyclic dependency of axis.';
33136   : sNcError := '33136 Function Block: Axis was not added to an axes group. Command is not valid.';
33151   : sNcError := '33151 State: Drive has invalid State.';
33153   : sNcError := '33153 Function Block: Gap control parameters invalid with current configuration.';
33154   : sNcError := '33154 Monitoring: Software position limit violation.';
33155   : sNcError := '33155 NC Programming: Target position is not reachable. No path available or target position unreachable.';
33157   : sNcError := '33157 NC Programming: Mover or relevant coordinates are busy.';
33158   : sNcError := '33158 NC Programming: A collision has occurred or would occur.';
33159   : sNcError := '33159 NC Programming: Invalid Track Specification. Geometric extension of this track is incompatible.';
33160   : sNcError := '33160 NC Programming: Command not allowed in track state.';
33161   : sNcError := '33161 Function Block: Invalid Reference passed to Function Block.';
33162   : sNcError := '33162 NC Programming: Path is locked against modifications.';
33164   : sNcError := '33164 Parameter: Position out of modulo range.';
33165   : sNcError := '33165 Parameter: Specified value AdditionalTurns at Options input is not allowed.';
33166   : sNcError := '33166 Function Block: Master/Slave sync position incompatible with sync direction.';
33169   : sNcError := '33169 State: Unexpected axis state. Axis error occurred after successful reset.';
33170   : sNcError := '33170 State: Invalid reference system.';
33171   : sNcError := '33171 State: Position not in reference system.';
33172   : sNcError := '33172 State: Previous command blocking execution.';
33176   : sNcError := '33176 Parameter: Invalid index.';
33177   : sNcError := '33177 Function Block: Command not allowed in current configuration.';
36655..36688 : sNcError := '36655-36688 Internal: Internal Error.';
36694   : sNcError := '36694 Internal: Internal Error.';
36697   : sNcError := '36697 Internal: Internal Error.';
36700..36706 : sNcError := '36700-36706 Internal: Internal Error.';
36709   : sNcError := '36709 Internal: Internal Error.';
36712..36814 : sNcError := '36712-36814 Internal: Internal Error.';
36816..36863 : sNcError := '36816-36863 Internal: Internal Error.';

ELSE
	sNcError := UDINT_TO_STRING(nNcError);
	sNcError := concat(sNcError, ' Unknown Error code');
END_CASE
END_ACTION

ACTION _state:

END_ACTION

END_FUNCTION_BLOCK

(* stored: Version 1.1.0.1, ProductVersion 3.1.4024.12
   POU FB_DriveDecoder: Id {0203e723-4504-0869-2058-544846f9f699}, SpecialFunc None
   Action _diag: Id {6a0391c1-a9a7-4fb6-b481-78d89c25331b}
   Action _ethercat: Id {d4aced07-e856-09b1-046b-f4f1db871967}
   Action _nc: Id {135acf2c-ae89-4dbc-9162-4c1dd2649f40}
   Action _state: Id {1f4cb215-1832-4de3-a21d-b29fc348d651} *)
